# EPICS substitutions: ek9000App/Db/EL1134.substitutions
file EL1134.template
{ 	pattern
	{
		TERMINAL,

	}
	{
	}
}
